	MoveL [[143.345,1275.593,0.000],[0.00000002,0.00000004,1.00000000,-0.00000004],[0,-1,0,0],rdkExtax], rdkSpeed, rdkZone, rdkTool, \WObj:=rdkWObj;
	MoveL [[133.284,1275.429,0.000],[0.00000002,0.00000004,1.00000000,-0.00000004],[0,-1,0,0],rdkExtax], rdkSpeed, rdkZone, rdkTool, \WObj:=rdkWObj;
	MoveL [[123.224,1275.245,0.000],[0.00000002,0.00000004,1.00000000,-0.00000004],[0,-1,0,0],rdkExtax], rdkSpeed, rdkZone, rdkTool, \WObj:=rdkWObj;
	MoveL [[113.164,1275.040,0.000],[0.00000002,0.00000004,1.00000000,-0.00000004],[0,-1,0,0],rdkExtax], rdkSpeed, rdkZone, rdkTool, \WObj:=rdkWObj;
	MoveL [[103.103,1274.816,0.000],[0.00000002,0.00000004,1.00000000,-0.00000004],[0,-1,0,0],rdkExtax], rdkSpeed, rdkZone, rdkTool, \WObj:=rdkWObj;
	MoveL [[93.043,1274.573,0.000],[0.00000002,0.00000004,1.00000000,-0.00000004],[0,-1,0,0],rdkExtax], rdkSpeed, rdkZone, rdkTool, \WObj:=rdkWObj;
	MoveL [[82.983,1274.311,0.000],[0.00000002,0.00000004,1.00000000,-0.00000004],[0,-1,0,0],rdkExtax], rdkSpeed, rdkZone, rdkTool, \WObj:=rdkWObj;
	MoveL [[72.922,1274.032,0.000],[0.00000002,0.00000004,1.00000000,-0.00000004],[0,-1,0,0],rdkExtax], rdkSpeed, rdkZone, rdkTool, \WObj:=rdkWObj;
	MoveL [[62.862,1273.736,0.000],[0.00000002,0.00000004,1.00000000,-0.00000004],[0,-1,0,0],rdkExtax], rdkSpeed, rdkZone, rdkTool, \WObj:=rdkWObj;
	MoveL [[52.801,1273.423,0.000],[0.00000002,0.00000004,1.00000000,-0.00000004],[0,-1,0,0],rdkExtax], rdkSpeed, rdkZone, rdkTool, \WObj:=rdkWObj;
	MoveL [[42.741,1273.094,0.000],[0.00000002,0.00000004,1.00000000,-0.00000004],[0,-1,0,0],rdkExtax], rdkSpeed, rdkZone, rdkTool, \WObj:=rdkWObj;
	MoveL [[32.680,1272.749,0.000],[0.00000002,0.00000004,1.00000000,-0.00000004],[0,-1,0,0],rdkExtax], rdkSpeed, rdkZone, rdkTool, \WObj:=rdkWObj;
	MoveL [[22.620,1272.390,0.000],[0.00000002,0.00000004,1.00000000,-0.00000004],[0,-1,0,0],rdkExtax], rdkSpeed, rdkZone, rdkTool, \WObj:=rdkWObj;
	MoveL [[16.560,1277.001,0.000],[0.00000002,0.00000004,1.00000000,-0.00000004],[0,-1,0,0],rdkExtax], rdkSpeed, rdkZone, rdkTool, \WObj:=rdkWObj;
	MoveL [[14.353,1286.214,0.000],[0.00000002,0.00000004,1.00000000,-0.00000004],[0,-1,0,0],rdkExtax], rdkSpeed, rdkZone, rdkTool, \WObj:=rdkWObj;
	MoveL [[12.501,1295.620,0.000],[0.00000002,0.00000004,1.00000000,-0.00000004],[0,-1,0,0],rdkExtax], rdkSpeed, rdkZone, rdkTool, \WObj:=rdkWObj;
	MoveL [[10.983,1305.202,0.000],[0.00000002,0.00000004,1.00000000,-0.00000004],[0,-1,0,0],rdkExtax], rdkSpeed, rdkZone, rdkTool, \WObj:=rdkWObj;
	MoveL [[9.778,1314.942,0.000],[0.00000002,0.00000004,1.00000000,-0.00000004],[0,-1,0,0],rdkExtax], rdkSpeed, rdkZone, rdkTool, \WObj:=rdkWObj;
	MoveL [[8.863,1324.822,0.000],[0.00000002,0.00000004,1.00000000,-0.00000004],[0,-1,0,0],rdkExtax], rdkSpeed, rdkZone, rdkTool, \WObj:=rdkWObj;
	MoveL [[8.219,1334.824,0.000],[0.00000002,0.00000004,1.00000000,-0.00000004],[0,-1,0,0],rdkExtax], rdkSpeed, rdkZone, rdkTool, \WObj:=rdkWObj;
	MoveL [[7.822,1344.931,0.000],[0.00000002,0.00000004,1.00000000,-0.00000004],[0,-1,0,0],rdkExtax], rdkSpeed, rdkZone, rdkTool, \WObj:=rdkWObj;
	MoveL [[7.652,1355.125,0.000],[0.00000002,0.00000004,1.00000000,-0.00000004],[0,-1,0,0],rdkExtax], rdkSpeed, rdkZone, rdkTool, \WObj:=rdkWObj;
	MoveL [[7.687,1365.387,0.000],[0.00000002,0.00000004,1.00000000,-0.00000004],[0,-1,0,0],rdkExtax], rdkSpeed, rdkZone, rdkTool, \WObj:=rdkWObj;
	MoveL [[7.907,1375.701,0.000],[0.00000002,0.00000004,1.00000000,-0.00000004],[0,-1,0,0],rdkExtax], rdkSpeed, rdkZone, rdkTool, \WObj:=rdkWObj;
	MoveL [[8.289,1386.047,0.000],[0.00000002,0.00000004,1.00000000,-0.00000004],[0,-1,0,0],rdkExtax], rdkSpeed, rdkZone, rdkTool, \WObj:=rdkWObj;
	MoveL [[8.812,1396.409,0.000],[0.00000002,0.00000004,1.00000000,-0.00000004],[0,-1,0,0],rdkExtax], rdkSpeed, rdkZone, rdkTool, \WObj:=rdkWObj;
	MoveL [[9.454,1406.769,0.000],[0.00000002,0.00000004,1.00000000,-0.00000004],[0,-1,0,0],rdkExtax], rdkSpeed, rdkZone, rdkTool, \WObj:=rdkWObj;
	MoveL [[10.195,1417.109,0.000],[0.00000002,0.00000004,1.00000000,-0.00000004],[0,-1,0,0],rdkExtax], rdkSpeed, rdkZone, rdkTool, \WObj:=rdkWObj;
	MoveL [[11.013,1427.410,0.000],[0.00000002,0.00000004,1.00000000,-0.00000004],[0,-1,0,0],rdkExtax], rdkSpeed, rdkZone, rdkTool, \WObj:=rdkWObj;
	MoveL [[11.886,1437.656,0.000],[0.00000002,0.00000004,1.00000000,-0.00000004],[0,-1,0,0],rdkExtax], rdkSpeed, rdkZone, rdkTool, \WObj:=rdkWObj;
	MoveL [[12.793,1447.828,0.000],[0.00000002,0.00000004,1.00000000,-0.00000004],[0,-1,0,0],rdkExtax], rdkSpeed, rdkZone, rdkTool, \WObj:=rdkWObj;
	MoveL [[13.713,1457.908,0.000],[0.00000002,0.00000004,1.00000000,-0.00000004],[0,-1,0,0],rdkExtax], rdkSpeed, rdkZone, rdkTool, \WObj:=rdkWObj;
	MoveL [[14.624,1467.879,0.000],[0.00000002,0.00000004,1.00000000,-0.00000004],[0,-1,0,0],rdkExtax], rdkSpeed, rdkZone, rdkTool, \WObj:=rdkWObj;
	MoveL [[15.505,1477.723,0.000],[0.00000002,0.00000004,1.00000000,-0.00000004],[0,-1,0,0],rdkExtax], rdkSpeed, rdkZone, rdkTool, \WObj:=rdkWObj;
	MoveL [[16.772,1487.917,0.000],[0.00000002,0.00000004,1.00000000,-0.00000004],[0,-1,0,0],rdkExtax], rdkSpeed, rdkZone, rdkTool, \WObj:=rdkWObj;
	MoveL [[18.876,1498.151,0.000],[0.00000002,0.00000004,1.00000000,-0.00000004],[0,-1,0,0],rdkExtax], rdkSpeed, rdkZone, rdkTool, \WObj:=rdkWObj;
	MoveL [[21.647,1508.050,0.000],[0.00000002,0.00000004,1.00000000,-0.00000004],[0,-1,0,0],rdkExtax], rdkSpeed, rdkZone, rdkTool, \WObj:=rdkWObj;
	MoveL [[25.057,1517.606,0.000],[0.00000002,0.00000004,1.00000000,-0.00000004],[0,-1,0,0],rdkExtax], rdkSpeed, rdkZone, rdkTool, \WObj:=rdkWObj;
	MoveL [[29.077,1526.811,0.000],[0.00000002,0.00000004,1.00000000,-0.00000004],[0,-1,0,0],rdkExtax], rdkSpeed, rdkZone, rdkTool, \WObj:=rdkWObj;
	MoveL [[33.677,1535.657,0.000],[0.00000002,0.00000004,1.00000000,-0.00000004],[0,-1,0,0],rdkExtax], rdkSpeed, rdkZone, rdkTool, \WObj:=rdkWObj;
	MoveL [[38.828,1544.135,0.000],[0.00000002,0.00000004,1.00000000,-0.00000004],[0,-1,0,0],rdkExtax], rdkSpeed, rdkZone, rdkTool, \WObj:=rdkWObj;
	MoveL [[44.502,1552.237,0.000],[0.00000002,0.00000004,1.00000000,-0.00000004],[0,-1,0,0],rdkExtax], rdkSpeed, rdkZone, rdkTool, \WObj:=rdkWObj;
	MoveL [[50.668,1559.956,0.000],[0.00000002,0.00000004,1.00000000,-0.00000004],[0,-1,0,0],rdkExtax], rdkSpeed, rdkZone, rdkTool, \WObj:=rdkWObj;
	MoveL [[57.299,1567.283,0.000],[0.00000002,0.00000004,1.00000000,-0.00000004],[0,-1,0,0],rdkExtax], rdkSpeed, rdkZone, rdkTool, \WObj:=rdkWObj;
	MoveL [[64.364,1574.209,0.000],[0.00000002,0.00000004,1.00000000,-0.00000004],[0,-1,0,0],rdkExtax], rdkSpeed, rdkZone, rdkTool, \WObj:=rdkWObj;
	MoveL [[71.835,1580.728,0.000],[0.00000002,0.00000004,1.00000000,-0.00000004],[0,-1,0,0],rdkExtax], rdkSpeed, rdkZone, rdkTool, \WObj:=rdkWObj;
	MoveL [[79.683,1586.830,0.000],[0.00000002,0.00000004,1.00000000,-0.00000004],[0,-1,0,0],rdkExtax], rdkSpeed, rdkZone, rdkTool, \WObj:=rdkWObj;
	MoveL [[87.878,1592.508,0.000],[0.00000002,0.00000004,1.00000000,-0.00000004],[0,-1,0,0],rdkExtax], rdkSpeed, rdkZone, rdkTool, \WObj:=rdkWObj;
	MoveL [[96.392,1597.753,0.000],[0.00000002,0.00000004,1.00000000,-0.00000004],[0,-1,0,0],rdkExtax], rdkSpeed, rdkZone, rdkTool, \WObj:=rdkWObj;
	MoveL [[105.194,1602.558,0.000],[0.00000002,0.00000004,1.00000000,-0.00000004],[0,-1,0,0],rdkExtax], rdkSpeed, rdkZone, rdkTool, \WObj:=rdkWObj;
	MoveL [[114.257,1606.914,0.000],[0.00000002,0.00000004,1.00000000,-0.00000004],[0,-1,0,0],rdkExtax], rdkSpeed, rdkZone, rdkTool, \WObj:=rdkWObj;
	MoveL [[123.551,1610.813,0.000],[0.00000002,0.00000004,1.00000000,-0.00000004],[0,-1,0,0],rdkExtax], rdkSpeed, rdkZone, rdkTool, \WObj:=rdkWObj;
	MoveL [[133.047,1614.246,0.000],[0.00000002,0.00000004,1.00000000,-0.00000004],[0,-1,0,0],rdkExtax], rdkSpeed, rdkZone, rdkTool, \WObj:=rdkWObj;
	MoveL [[142.716,1617.207,0.000],[0.00000002,0.00000004,1.00000000,-0.00000004],[0,-1,0,0],rdkExtax], rdkSpeed, rdkZone, rdkTool, \WObj:=rdkWObj;
	MoveL [[152.528,1619.686,0.000],[0.00000002,0.00000004,1.00000000,-0.00000004],[0,-1,0,0],rdkExtax], rdkSpeed, rdkZone, rdkTool, \WObj:=rdkWObj;
	MoveL [[162.454,1621.675,0.000],[0.00000002,0.00000004,1.00000000,-0.00000004],[0,-1,0,0],rdkExtax], rdkSpeed, rdkZone, rdkTool, \WObj:=rdkWObj;
	MoveL [[172.466,1623.167,0.000],[0.00000002,0.00000004,1.00000000,-0.00000004],[0,-1,0,0],rdkExtax], rdkSpeed, rdkZone, rdkTool, \WObj:=rdkWObj;
	MoveL [[182.535,1624.153,0.000],[0.00000002,0.00000004,1.00000000,-0.00000004],[0,-1,0,0],rdkExtax], rdkSpeed, rdkZone, rdkTool, \WObj:=rdkWObj;
	MoveL [[192.630,1624.625,0.000],[0.00000002,0.00000004,1.00000000,-0.00000004],[0,-1,0,0],rdkExtax], rdkSpeed, rdkZone, rdkTool, \WObj:=rdkWObj;
	MoveL [[191.948,1521.248,0.000],[0.00000002,0.00000004,1.00000000,-0.00000004],[0,-1,0,0],rdkExtax], rdkSpeed, rdkZone, rdkTool, \WObj:=rdkWObj;
	MoveL [[181.490,1520.957,0.000],[0.00000002,0.00000004,1.00000000,-0.00000004],[0,-1,0,0],rdkExtax], rdkSpeed, rdkZone, rdkTool, \WObj:=rdkWObj;
	MoveL [[171.373,1519.493,0.000],[0.00000002,0.00000004,1.00000000,-0.00000004],[0,-1,0,0],rdkExtax], rdkSpeed, rdkZone, rdkTool, \WObj:=rdkWObj;
	MoveL [[161.642,1516.933,0.000],[0.00000002,0.00000004,1.00000000,-0.00000004],[0,-1,0,0],rdkExtax], rdkSpeed, rdkZone, rdkTool, \WObj:=rdkWObj;
	MoveL [[152.344,1513.350,0.000],[0.00000002,0.00000004,1.00000000,-0.00000004],[0,-1,0,0],rdkExtax], rdkSpeed, rdkZone, rdkTool, \WObj:=rdkWObj;
	MoveL [[143.525,1508.821,0.000],[0.00000002,0.00000004,1.00000000,-0.00000004],[0,-1,0,0],rdkExtax], rdkSpeed, rdkZone, rdkTool, \WObj:=rdkWObj;
	MoveL [[135.231,1503.420,0.000],[0.00000002,0.00000004,1.00000000,-0.00000004],[0,-1,0,0],rdkExtax], rdkSpeed, rdkZone, rdkTool, \WObj:=rdkWObj;
	MoveL [[127.510,1497.222,0.000],[0.00000002,0.00000004,1.00000000,-0.00000004],[0,-1,0,0],rdkExtax], rdkSpeed, rdkZone, rdkTool, \WObj:=rdkWObj;
	MoveL [[120.406,1490.303,0.000],[0.00000002,0.00000004,1.00000000,-0.00000004],[0,-1,0,0],rdkExtax], rdkSpeed, rdkZone, rdkTool, \WObj:=rdkWObj;
	MoveL [[113.967,1482.738,0.000],[0.00000002,0.00000004,1.00000000,-0.00000004],[0,-1,0,0],rdkExtax], rdkSpeed, rdkZone, rdkTool, \WObj:=rdkWObj;
	MoveL [[108.239,1474.601,0.000],[0.00000002,0.00000004,1.00000000,-0.00000004],[0,-1,0,0],rdkExtax], rdkSpeed, rdkZone, rdkTool, \WObj:=rdkWObj;
	MoveL [[103.267,1465.968,0.000],[0.00000002,0.00000004,1.00000000,-0.00000004],[0,-1,0,0],rdkExtax], rdkSpeed, rdkZone, rdkTool, \WObj:=rdkWObj;
	MoveL [[99.099,1456.914,0.000],[0.00000002,0.00000004,1.00000000,-0.00000004],[0,-1,0,0],rdkExtax], rdkSpeed, rdkZone, rdkTool, \WObj:=rdkWObj;
	MoveL [[95.780,1447.514,0.000],[0.00000002,0.00000004,1.00000000,-0.00000004],[0,-1,0,0],rdkExtax], rdkSpeed, rdkZone, rdkTool, \WObj:=rdkWObj;
	MoveL [[93.357,1437.843,0.000],[0.00000002,0.00000004,1.00000000,-0.00000004],[0,-1,0,0],rdkExtax], rdkSpeed, rdkZone, rdkTool, \WObj:=rdkWObj;
	MoveL [[91.876,1427.977,0.000],[0.00000002,0.00000004,1.00000000,-0.00000004],[0,-1,0,0],rdkExtax], rdkSpeed, rdkZone, rdkTool, \WObj:=rdkWObj;
	MoveL [[91.384,1417.990,0.000],[0.00000002,0.00000004,1.00000000,-0.00000004],[0,-1,0,0],rdkExtax], rdkSpeed, rdkZone, rdkTool, \WObj:=rdkWObj;
	MoveL [[91.927,1407.958,0.000],[0.00000002,0.00000004,1.00000000,-0.00000004],[0,-1,0,0],rdkExtax], rdkSpeed, rdkZone, rdkTool, \WObj:=rdkWObj;
	MoveL [[93.550,1397.955,0.000],[0.00000002,0.00000004,1.00000000,-0.00000004],[0,-1,0,0],rdkExtax], rdkSpeed, rdkZone, rdkTool, \WObj:=rdkWObj;
	MoveL [[96.301,1388.057,0.000],[0.00000002,0.00000004,1.00000000,-0.00000004],[0,-1,0,0],rdkExtax], rdkSpeed, rdkZone, rdkTool, \WObj:=rdkWObj;
	MoveL [[101.782,1381.318,0.000],[0.00000002,0.00000004,1.00000000,-0.00000004],[0,-1,0,0],rdkExtax], rdkSpeed, rdkZone, rdkTool, \WObj:=rdkWObj;
	MoveL [[111.384,1381.237,0.000],[0.00000002,0.00000004,1.00000000,-0.00000004],[0,-1,0,0],rdkExtax], rdkSpeed, rdkZone, rdkTool, \WObj:=rdkWObj;
	MoveL [[121.241,1380.943,0.000],[0.00000002,0.00000004,1.00000000,-0.00000004],[0,-1,0,0],rdkExtax], rdkSpeed, rdkZone, rdkTool, \WObj:=rdkWObj;
	MoveL [[131.317,1380.480,0.000],[0.00000002,0.00000004,1.00000000,-0.00000004],[0,-1,0,0],rdkExtax], rdkSpeed, rdkZone, rdkTool, \WObj:=rdkWObj;
	MoveL [[141.577,1379.891,0.000],[0.00000002,0.00000004,1.00000000,-0.00000004],[0,-1,0,0],rdkExtax], rdkSpeed, rdkZone, rdkTool, \WObj:=rdkWObj;
	MoveL [[151.984,1379.219,0.000],[0.00000002,0.00000004,1.00000000,-0.00000004],[0,-1,0,0],rdkExtax], rdkSpeed, rdkZone, rdkTool, \WObj:=rdkWObj;
	MoveL [[162.504,1378.508,0.000],[0.00000002,0.00000004,1.00000000,-0.00000004],[0,-1,0,0],rdkExtax], rdkSpeed, rdkZone, rdkTool, \WObj:=rdkWObj;
	MoveL [[173.101,1377.802,0.000],[0.00000002,0.00000004,1.00000000,-0.00000004],[0,-1,0,0],rdkExtax], rdkSpeed, rdkZone, rdkTool, \WObj:=rdkWObj;
	MoveL [[183.740,1377.143,0.000],[0.00000002,0.00000004,1.00000000,-0.00000004],[0,-1,0,0],rdkExtax], rdkSpeed, rdkZone, rdkTool, \WObj:=rdkWObj;
	MoveL [[194.385,1376.575,0.000],[0.00000002,0.00000004,1.00000000,-0.00000004],[0,-1,0,0],rdkExtax], rdkSpeed, rdkZone, rdkTool, \WObj:=rdkWObj;
	MoveL [[205.000,1376.141,0.000],[0.00000002,0.00000004,1.00000000,-0.00000004],[0,-1,0,0],rdkExtax], rdkSpeed, rdkZone, rdkTool, \WObj:=rdkWObj;
	MoveL [[215.551,1375.885,0.000],[0.00000002,0.00000004,1.00000000,-0.00000004],[0,-1,0,0],rdkExtax], rdkSpeed, rdkZone, rdkTool, \WObj:=rdkWObj;
	MoveL [[226.001,1375.850,0.000],[0.00000002,0.00000004,1.00000000,-0.00000004],[0,-1,0,0],rdkExtax], rdkSpeed, rdkZone, rdkTool, \WObj:=rdkWObj;
	MoveL [[236.316,1376.080,0.000],[0.00000002,0.00000004,1.00000000,-0.00000004],[0,-1,0,0],rdkExtax], rdkSpeed, rdkZone, rdkTool, \WObj:=rdkWObj;
	MoveL [[246.459,1376.617,0.000],[0.00000002,0.00000004,1.00000000,-0.00000004],[0,-1,0,0],rdkExtax], rdkSpeed, rdkZone, rdkTool, \WObj:=rdkWObj;
	MoveL [[256.395,1377.506,0.000],[0.00000002,0.00000004,1.00000000,-0.00000004],[0,-1,0,0],rdkExtax], rdkSpeed, rdkZone, rdkTool, \WObj:=rdkWObj;
	MoveL [[266.090,1378.789,0.000],[0.00000002,0.00000004,1.00000000,-0.00000004],[0,-1,0,0],rdkExtax], rdkSpeed, rdkZone, rdkTool, \WObj:=rdkWObj;
	MoveL [[275.506,1380.510,0.000],[0.00000002,0.00000004,1.00000000,-0.00000004],[0,-1,0,0],rdkExtax], rdkSpeed, rdkZone, rdkTool, \WObj:=rdkWObj;
	MoveL [[284.610,1382.713,0.000],[0.00000002,0.00000004,1.00000000,-0.00000004],[0,-1,0,0],rdkExtax], rdkSpeed, rdkZone, rdkTool, \WObj:=rdkWObj;
	MoveL [[293.364,1385.440,0.000],[0.00000002,0.00000004,1.00000000,-0.00000004],[0,-1,0,0],rdkExtax], rdkSpeed, rdkZone, rdkTool, \WObj:=rdkWObj;
	MoveL [[301.735,1388.735,0.000],[0.00000002,0.00000004,1.00000000,-0.00000004],[0,-1,0,0],rdkExtax], rdkSpeed, rdkZone, rdkTool, \WObj:=rdkWObj;
	MoveL [[305.438,1397.949,0.000],[0.00000002,0.00000004,1.00000000,-0.00000004],[0,-1,0,0],rdkExtax], rdkSpeed, rdkZone, rdkTool, \WObj:=rdkWObj;
	MoveL [[307.003,1408.567,0.000],[0.00000002,0.00000004,1.00000000,-0.00000004],[0,-1,0,0],rdkExtax], rdkSpeed, rdkZone, rdkTool, \WObj:=rdkWObj;
	MoveL [[307.559,1419.010,0.000],[0.00000002,0.00000004,1.00000000,-0.00000004],[0,-1,0,0],rdkExtax], rdkSpeed, rdkZone, rdkTool, \WObj:=rdkWObj;
	MoveL [[307.145,1429.225,0.000],[0.00000002,0.00000004,1.00000000,-0.00000004],[0,-1,0,0],rdkExtax], rdkSpeed, rdkZone, rdkTool, \WObj:=rdkWObj;
	MoveL [[305.794,1439.164,0.000],[0.00000002,0.00000004,1.00000000,-0.00000004],[0,-1,0,0],rdkExtax], rdkSpeed, rdkZone, rdkTool, \WObj:=rdkWObj;
	MoveL [[303.543,1448.776,0.000],[0.00000002,0.00000004,1.00000000,-0.00000004],[0,-1,0,0],rdkExtax], rdkSpeed, rdkZone, rdkTool, \WObj:=rdkWObj;
	MoveL [[300.427,1458.011,0.000],[0.00000002,0.00000004,1.00000000,-0.00000004],[0,-1,0,0],rdkExtax], rdkSpeed, rdkZone, rdkTool, \WObj:=rdkWObj;
	MoveL [[296.482,1466.819,0.000],[0.00000002,0.00000004,1.00000000,-0.00000004],[0,-1,0,0],rdkExtax], rdkSpeed, rdkZone, rdkTool, \WObj:=rdkWObj;
	MoveL [[291.744,1475.149,0.000],[0.00000002,0.00000004,1.00000000,-0.00000004],[0,-1,0,0],rdkExtax], rdkSpeed, rdkZone, rdkTool, \WObj:=rdkWObj;
	MoveL [[286.249,1482.952,0.000],[0.00000002,0.00000004,1.00000000,-0.00000004],[0,-1,0,0],rdkExtax], rdkSpeed, rdkZone, rdkTool, \WObj:=rdkWObj;
	MoveL [[280.032,1490.176,0.000],[0.00000002,0.00000004,1.00000000,-0.00000004],[0,-1,0,0],rdkExtax], rdkSpeed, rdkZone, rdkTool, \WObj:=rdkWObj;
	MoveL [[273.129,1496.773,0.000],[0.00000002,0.00000004,1.00000000,-0.00000004],[0,-1,0,0],rdkExtax], rdkSpeed, rdkZone, rdkTool, \WObj:=rdkWObj;
	MoveL [[265.575,1502.691,0.000],[0.00000002,0.00000004,1.00000000,-0.00000004],[0,-1,0,0],rdkExtax], rdkSpeed, rdkZone, rdkTool, \WObj:=rdkWObj;
	MoveL [[257.407,1507.881,0.000],[0.00000002,0.00000004,1.00000000,-0.00000004],[0,-1,0,0],rdkExtax], rdkSpeed, rdkZone, rdkTool, \WObj:=rdkWObj;
	MoveL [[248.660,1512.292,0.000],[0.00000002,0.00000004,1.00000000,-0.00000004],[0,-1,0,0],rdkExtax], rdkSpeed, rdkZone, rdkTool, \WObj:=rdkWObj;
	MoveL [[239.369,1515.875,0.000],[0.00000002,0.00000004,1.00000000,-0.00000004],[0,-1,0,0],rdkExtax], rdkSpeed, rdkZone, rdkTool, \WObj:=rdkWObj;
	MoveL [[229.571,1518.578,0.000],[0.00000002,0.00000004,1.00000000,-0.00000004],[0,-1,0,0],rdkExtax], rdkSpeed, rdkZone, rdkTool, \WObj:=rdkWObj;
	MoveL [[219.301,1520.353,0.000],[0.00000002,0.00000004,1.00000000,-0.00000004],[0,-1,0,0],rdkExtax], rdkSpeed, rdkZone, rdkTool, \WObj:=rdkWObj;
	MoveL [[208.595,1521.148,0.000],[0.00000002,0.00000004,1.00000000,-0.00000004],[0,-1,0,0],rdkExtax], rdkSpeed, rdkZone, rdkTool, \WObj:=rdkWObj;
	MoveL [[197.489,1520.913,0.000],[0.00000002,0.00000004,1.00000000,-0.00000004],[0,-1,0,0],rdkExtax], rdkSpeed, rdkZone, rdkTool, \WObj:=rdkWObj;
	MoveL [[197.489,1520.913,100.000],[0.00000002,0.00000004,1.00000000,-0.00000004],[0,-1,0,0],rdkExtax], rdkSpeed, rdkZone, rdkTool, \WObj:=rdkWObj;
	MoveL [[374.392,2000.149,100.000],[0.00000002,0.00000004,1.00000000,-0.00000004],[0,-1,0,0],rdkExtax], rdkSpeed, rdkZone, rdkTool, \WObj:=rdkWObj;
	TPWrite "Drawing path3000";
	SetColorRGB(0.643,0.071,0.000);
	MoveL [[374.392,2000.149,0.000],[0.00000002,0.00000004,1.00000000,-0.00000004],[0,-1,0,0],rdkExtax], rdkSpeed, rdkZone, rdkTool, \WObj:=rdkWObj;
	MoveL [[380.983,1992.390,0.000],[0.00000002,0.00000004,1.00000000,-0.00000004],[0,-1,0,0],rdkExtax], rdkSpeed, rdkZone, rdkTool, \WObj:=rdkWObj;
	MoveL [[386.344,1984.065,0.000],[0.00000002,0.00000004,1.00000000,-0.00000004],[0,-1,0,0],rdkExtax], rdkSpeed, rdkZone, rdkTool, \WObj:=rdkWObj;
	MoveL [[390.508,1975.269,0.000],[0.00000002,0.00000004,1.00000000,-0.00000004],[0,-1,0,0],rdkExtax], rdkSpeed, rdkZone, rdkTool, \WObj:=rdkWObj;
	MoveL [[393.510,1966.101,0.000],[0.00000002,0.00000004,1.00000000,-0.00000004],[0,-1,0,0],rdkExtax], rdkSpeed, rdkZone, rdkTool, \WObj:=rdkWObj;
	MoveL [[395.384,1956.658,0.000],[0.00000002,0.00000004,1.00000000,-0.00000004],[0,-1,0,0],rdkExtax], rdkSpeed, rdkZone, rdkTool, \WObj:=rdkWObj;
	MoveL [[396.164,1947.037,0.000],[0.00000002,0.00000004,1.00000000,-0.00000004],[0,-1,0,0],rdkExtax], rdkSpeed, rdkZone, rdkTool, \WObj:=rdkWObj;
	MoveL [[395.885,1937.335,0.000],[0.00000002,0.00000004,1.00000000,-0.00000004],[0,-1,0,0],rdkExtax], rdkSpeed, rdkZone, rdkTool, \WObj:=rdkWObj;
	MoveL [[394.580,1927.650,0.000],[0.00000002,0.00000004,1.00000000,-0.00000004],[0,-1,0,0],rdkExtax], rdkSpeed, rdkZone, rdkTool, \WObj:=rdkWObj;
	MoveL [[392.283,1918.079,0.000],[0.00000002,0.00000004,1.00000000,-0.00000004],[0,-1,0,0],rdkExtax], rdkSpeed, rdkZone, rdkTool, \WObj:=rdkWObj;
	MoveL [[389.030,1908.719,0.000],[0.00000002,0.00000004,1.00000000,-0.00000004],[0,-1,0,0],rdkExtax], rdkSpeed, rdkZone, rdkTool, \WObj:=rdkWObj;
	MoveL [[384.853,1899.669,0.000],[0.00000002,0.00000004,1.00000000,-0.00000004],[0,-1,0,0],rdkExtax], rdkSpeed, rdkZone, rdkTool, \WObj:=rdkWObj;
	MoveL [[379.788,1891.024,0.000],[0.00000002,0.00000004,1.00000000,-0.00000004],[0,-1,0,0],rdkExtax], rdkSpeed, rdkZone, rdkTool, \WObj:=rdkWObj;
	MoveL [[373.868,1882.883,0.000],[0.00000002,0.00000004,1.00000000,-0.00000004],[0,-1,0,0],rdkExtax], rdkSpeed, rdkZone, rdkTool, \WObj:=rdkWObj;
	MoveL [[367.127,1875.342,0.000],[0.00000002,0.00000004,1.00000000,-0.00000004],[0,-1,0,0],rdkExtax], rdkSpeed, rdkZone, rdkTool, \WObj:=rdkWObj;
	MoveL [[359.601,1868.499,0.000],[0.00000002,0.00000004,1.00000000,-0.00000004],[0,-1,0,0],rdkExtax], rdkSpeed, rdkZone, rdkTool, \WObj:=rdkWObj;
	MoveL [[351.322,1862.452,0.000],[0.00000002,0.00000004,1.00000000,-0.00000004],[0,-1,0,0],rdkExtax], rdkSpeed, rdkZone, rdkTool, \WObj:=rdkWObj;
	MoveL [[342.325,1857.297,0.000],[0.00000002,0.00000004,1.00000000,-0.00000004],[0,-1,0,0],rdkExtax], rdkSpeed, rdkZone, rdkTool, \WObj:=rdkWObj;
	MoveL [[332.645,1853.133,0.000],[0.00000002,0.00000004,1.00000000,-0.00000004],[0,-1,0,0],rdkExtax], rdkSpeed, rdkZone, rdkTool, \WObj:=rdkWObj;
	MoveL [[322.314,1850.055,0.000],[0.00000002,0.00000004,1.00000000,-0.00000004],[0,-1,0,0],rdkExtax], rdkSpeed, rdkZone, rdkTool, \WObj:=rdkWObj;
	MoveL [[311.202,1847.909,0.000],[0.00000002,0.00000004,1.00000000,-0.00000004],[0,-1,0,0],rdkExtax], rdkSpeed, rdkZone, rdkTool, \WObj:=rdkWObj;
	MoveL [[299.905,1844.582,0.000],[0.00000002,0.00000004,1.00000000,-0.00000004],[0,-1,0,0],rdkExtax], rdkSpeed, rdkZone, rdkTool, \WObj:=rdkWObj;
	MoveL [[289.209,1839.822,0.000],[0.00000002,0.00000004,1.00000000,-0.00000004],[0,-1,0,0],rdkExtax], rdkSpeed, rdkZone, rdkTool, \WObj:=rdkWObj;
	MoveL [[279.340,1833.918,0.000],[0.00000002,0.00000004,1.00000000,-0.00000004],[0,-1,0,0],rdkExtax], rdkSpeed, rdkZone, rdkTool, \WObj:=rdkWObj;
	MoveL [[270.524,1827.156,0.000],[0.00000002,0.00000004,1.00000000,-0.00000004],[0,-1,0,0],rdkExtax], rdkSpeed, rdkZone, rdkTool, \WObj:=rdkWObj;
	MoveL [[262.987,1819.826,0.000],[0.00000002,0.00000004,1.00000000,-0.00000004],[0,-1,0,0],rdkExtax], rdkSpeed, rdkZone, rdkTool, \WObj:=rdkWObj;
	MoveL [[256.956,1812.214,0.000],[0.00000002,0.00000004,1.00000000,-0.00000004],[0,-1,0,0],rdkExtax], rdkSpeed, rdkZone, rdkTool, \WObj:=rdkWObj;
	MoveL [[252.657,1804.611,0.000],[0.00000002,0.00000004,1.00000000,-0.00000004],[0,-1,0,0],rdkExtax], rdkSpeed, rdkZone, rdkTool, \WObj:=rdkWObj;
	MoveL [[250.316,1797.302,0.000],[0.00000002,0.00000004,1.00000000,-0.00000004],[0,-1,0,0],rdkExtax], rdkSpeed, rdkZone, rdkTool, \WObj:=rdkWObj;
	MoveL [[250.159,1790.578,0.000],[0.00000002,0.00000004,1.00000000,-0.00000004],[0,-1,0,0],rdkExtax], rdkSpeed, rdkZone, rdkTool, \WObj:=rdkWObj;
	MoveL [[252.412,1784.725,0.000],[0.00000002,0.00000004,1.00000000,-0.00000004],[0,-1,0,0],rdkExtax], rdkSpeed, rdkZone, rdkTool, \WObj:=rdkWObj;
	MoveL [[257.302,1780.031,0.000],[0.00000002,0.00000004,1.00000000,-0.00000004],[0,-1,0,0],rdkExtax], rdkSpeed, rdkZone, rdkTool, \WObj:=rdkWObj;
	MoveL [[265.055,1776.786,0.000],[0.00000002,0.00000004,1.00000000,-0.00000004],[0,-1,0,0],rdkExtax], rdkSpeed, rdkZone, rdkTool, \WObj:=rdkWObj;
	MoveL [[275.896,1775.276,0.000],[0.00000002,0.00000004,1.00000000,-0.00000004],[0,-1,0,0],rdkExtax], rdkSpeed, rdkZone, rdkTool, \WObj:=rdkWObj;
	MoveL [[290.052,1775.790,0.000],[0.00000002,0.00000004,1.00000000,-0.00000004],[0,-1,0,0],rdkExtax], rdkSpeed, rdkZone, rdkTool, \WObj:=rdkWObj;
	MoveL [[303.834,1777.432,0.000],[0.00000002,0.00000004,1.00000000,-0.00000004],[0,-1,0,0],rdkExtax], rdkSpeed, rdkZone, rdkTool, \WObj:=rdkWObj;
	MoveL [[314.296,1778.411,0.000],[0.00000002,0.00000004,1.00000000,-0.00000004],[0,-1,0,0],rdkExtax], rdkSpeed, rdkZone, rdkTool, \WObj:=rdkWObj;
	MoveL [[325.048,1779.340,0.000],[0.00000002,0.00000004,1.00000000,-0.00000004],[0,-1,0,0],rdkExtax], rdkSpeed, rdkZone, rdkTool, \WObj:=rdkWObj;
	MoveL [[335.852,1780.022,0.000],[0.00000002,0.00000004,1.00000000,-0.00000004],[0,-1,0,0],rdkExtax], rdkSpeed, rdkZone, rdkTool, \WObj:=rdkWObj;
	MoveL [[346.467,1780.260,0.000],[0.00000002,0.00000004,1.00000000,-0.00000004],[0,-1,0,0],rdkExtax], rdkSpeed, rdkZone, rdkTool, \WObj:=rdkWObj;
	MoveL [[356.655,1779.857,0.000],[0.00000002,0.00000004,1.00000000,-0.00000004],[0,-1,0,0],rdkExtax], rdkSpeed, rdkZone, rdkTool, \WObj:=rdkWObj;
	MoveL [[366.177,1778.616,0.000],[0.00000002,0.00000004,1.00000000,-0.00000004],[0,-1,0,0],rdkExtax], rdkSpeed, rdkZone, rdkTool, \WObj:=rdkWObj;
	MoveL [[374.793,1776.339,0.000],[0.00000002,0.00000004,1.00000000,-0.00000004],[0,-1,0,0],rdkExtax], rdkSpeed, rdkZone, rdkTool, \WObj:=rdkWObj;
	MoveL [[382.264,1772.830,0.000],[0.00000002,0.00000004,1.00000000,-0.00000004],[0,-1,0,0],rdkExtax], rdkSpeed, rdkZone, rdkTool, \WObj:=rdkWObj;
	MoveL [[388.351,1767.892,0.000],[0.00000002,0.00000004,1.00000000,-0.00000004],[0,-1,0,0],rdkExtax], rdkSpeed, rdkZone, rdkTool, \WObj:=rdkWObj;
	MoveL [[392.816,1761.327,0.000],[0.00000002,0.00000004,1.00000000,-0.00000004],[0,-1,0,0],rdkExtax], rdkSpeed, rdkZone, rdkTool, \WObj:=rdkWObj;
	MoveL [[395.418,1752.940,0.000],[0.00000002,0.00000004,1.00000000,-0.00000004],[0,-1,0,0],rdkExtax], rdkSpeed, rdkZone, rdkTool, \WObj:=rdkWObj;
	MoveL [[395.918,1742.532,0.000],[0.00000002,0.00000004,1.00000000,-0.00000004],[0,-1,0,0],rdkExtax], rdkSpeed, rdkZone, rdkTool, \WObj:=rdkWObj;
	MoveL [[394.078,1729.906,0.000],[0.00000002,0.00000004,1.00000000,-0.00000004],[0,-1,0,0],rdkExtax], rdkSpeed, rdkZone, rdkTool, \WObj:=rdkWObj;
	MoveL [[392.731,1715.600,0.000],[0.00000002,0.00000004,1.00000000,-0.00000004],[0,-1,0,0],rdkExtax], rdkSpeed, rdkZone, rdkTool, \WObj:=rdkWObj;
	MoveL [[393.844,1703.189,0.000],[0.00000002,0.00000004,1.00000000,-0.00000004],[0,-1,0,0],rdkExtax], rdkSpeed, rdkZone, rdkTool, \WObj:=rdkWObj;
	MoveL [[393.047,1692.845,0.000],[0.00000002,0.00000004,1.00000000,-0.00000004],[0,-1,0,0],rdkExtax], rdkSpeed, rdkZone, rdkTool, \WObj:=rdkWObj;
	MoveL [[390.495,1684.403,0.000],[0.00000002,0.00000004,1.00000000,-0.00000004],[0,-1,0,0],rdkExtax], rdkSpeed, rdkZone, rdkTool, \WObj:=rdkWObj;
	MoveL [[386.347,1677.698,0.000],[0.00000002,0.00000004,1.00000000,-0.00000004],[0,-1,0,0],rdkExtax], rdkSpeed, rdkZone, rdkTool, \WObj:=rdkWObj;
	MoveL [[380.758,1672.565,0.000],[0.00000002,0.00000004,1.00000000,-0.00000004],[0,-1,0,0],rdkExtax], rdkSpeed, rdkZone, rdkTool, \WObj:=rdkWObj;
	MoveL [[373.886,1668.838,0.000],[0.00000002,0.00000004,1.00000000,-0.00000004],[0,-1,0,0],rdkExtax], rdkSpeed, rdkZone, rdkTool, \WObj:=rdkWObj;
	MoveL [[365.887,1666.354,0.000],[0.00000002,0.00000004,1.00000000,-0.00000004],[0,-1,0,0],rdkExtax], rdkSpeed, rdkZone, rdkTool, \WObj:=rdkWObj;
	MoveL [[356.917,1664.946,0.000],[0.00000002,0.00000004,1.00000000,-0.00000004],[0,-1,0,0],rdkExtax], rdkSpeed, rdkZone, rdkTool, \WObj:=rdkWObj;
	MoveL [[347.135,1664.451,0.000],[0.00000002,0.00000004,1.00000000,-0.00000004],[0,-1,0,0],rdkExtax], rdkSpeed, rdkZone, rdkTool, \WObj:=rdkWObj;
	MoveL [[336.696,1664.702,0.000],[0.00000002,0.00000004,1.00000000,-0.00000004],[0,-1,0,0],rdkExtax], rdkSpeed, rdkZone, rdkTool, \WObj:=rdkWObj;
	MoveL [[325.758,1665.535,0.000],[0.00000002,0.00000004,1.00000000,-0.00000004],[0,-1,0,0],rdkExtax], rdkSpeed, rdkZone, rdkTool, \WObj:=rdkWObj;
	MoveL [[314.476,1666.785,0.000],[0.00000002,0.00000004,1.00000000,-0.00000004],[0,-1,0,0],rdkExtax], rdkSpeed, rdkZone, rdkTool, \WObj:=rdkWObj;
	MoveL [[303.008,1668.286,0.000],[0.00000002,0.00000004,1.00000000,-0.00000004],[0,-1,0,0],rdkExtax], rdkSpeed, rdkZone, rdkTool, \WObj:=rdkWObj;
	MoveL [[291.511,1669.874,0.000],[0.00000002,0.00000004,1.00000000,-0.00000004],[0,-1,0,0],rdkExtax], rdkSpeed, rdkZone, rdkTool, \WObj:=rdkWObj;
	MoveL [[280.141,1671.384,0.000],[0.00000002,0.00000004,1.00000000,-0.00000004],[0,-1,0,0],rdkExtax], rdkSpeed, rdkZone, rdkTool, \WObj:=rdkWObj;
	MoveL [[269.055,1672.650,0.000],[0.00000002,0.00000004,1.00000000,-0.00000004],[0,-1,0,0],rdkExtax], rdkSpeed, rdkZone, rdkTool, \WObj:=rdkWObj;
	MoveL [[258.410,1673.508,0.000],[0.00000002,0.00000004,1.00000000,-0.00000004],[0,-1,0,0],rdkExtax], rdkSpeed, rdkZone, rdkTool, \WObj:=rdkWObj;
	MoveL [[248.363,1673.792,0.000],[0.00000002,0.00000004,1.00000000,-0.00000004],[0,-1,0,0],rdkExtax], rdkSpeed, rdkZone, rdkTool, \WObj:=rdkWObj;
	MoveL [[239.070,1673.338,0.000],[0.00000002,0.00000004,1.00000000,-0.00000004],[0,-1,0,0],rdkExtax], rdkSpeed, rdkZone, rdkTool, \WObj:=rdkWObj;
	MoveL [[230.688,1671.981,0.000],[0.00000002,0.00000004,1.00000000,-0.00000004],[0,-1,0,0],rdkExtax], rdkSpeed, rdkZone, rdkTool, \WObj:=rdkWObj;
	MoveL [[220.678,1672.266,0.000],[0.00000002,0.00000004,1.00000000,-0.00000004],[0,-1,0,0],rdkExtax], rdkSpeed, rdkZone, rdkTool, \WObj:=rdkWObj;
	MoveL [[210.627,1672.439,0.000],[0.00000002,0.00000004,1.00000000,-0.00000004],[0,-1,0,0],rdkExtax], rdkSpeed, rdkZone, rdkTool, \WObj:=rdkWObj;
	MoveL [[200.572,1672.480,0.000],[0.00000002,0.00000004,1.00000000,-0.00000004],[0,-1,0,0],rdkExtax], rdkSpeed, rdkZone, rdkTool, \WObj:=rdkWObj;
	MoveL [[190.513,1672.402,0.000],[0.00000002,0.00000004,1.00000000,-0.00000004],[0,-1,0,0],rdkExtax], rdkSpeed, rdkZone, rdkTool, \WObj:=rdkWObj;
	MoveL [[180.452,1672.223,0.000],[0.00000002,0.00000004,1.00000000,-0.00000004],[0,-1,0,0],rdkExtax], rdkSpeed, rdkZone, rdkTool, \WObj:=rdkWObj;
	MoveL [[170.388,1671.956,0.000],[0.00000002,0.00000004,1.00000000,-0.00000004],[0,-1,0,0],rdkExtax], rdkSpeed, rdkZone, rdkTool, \WObj:=rdkWObj;
	MoveL [[160.323,1671.617,0.000],[0.00000002,0.00000004,1.00000000,-0.00000004],[0,-1,0,0],rdkExtax], rdkSpeed, rdkZone, rdkTool, \WObj:=rdkWObj;
	MoveL [[150.258,1671.223,0.000],[0.00000002,0.00000004,1.00000000,-0.00000004],[0,-1,0,0],rdkExtax], rdkSpeed, rdkZone, rdkTool, \WObj:=rdkWObj;
	MoveL [[140.193,1670.787,0.000],[0.00000002,0.00000004,1.00000000,-0.00000004],[0,-1,0,0],rdkExtax], rdkSpeed, rdkZone, rdkTool, \WObj:=rdkWObj;
	MoveL [[130.128,1670.327,0.000],[0.00000002,0.00000004,1.00000000,-0.00000004],[0,-1,0,0],rdkExtax], rdkSpeed, rdkZone, rdkTool, \WObj:=rdkWObj;
	MoveL [[120.066,1669.856,0.000],[0.00000002,0.00000004,1.00000000,-0.00000004],[0,-1,0,0],rdkExtax], rdkSpeed, rdkZone, rdkTool, \WObj:=rdkWObj;
	MoveL [[110.006,1669.390,0.000],[0.00000002,0.00000004,1.00000000,-0.00000004],[0,-1,0,0],rdkExtax], rdkSpeed, rdkZone, rdkTool, \WObj:=rdkWObj;
	MoveL [[99.949,1668.946,0.000],[0.00000002,0.00000004,1.00000000,-0.00000004],[0,-1,0,0],rdkExtax], rdkSpeed, rdkZone, rdkTool, \WObj:=rdkWObj;
	MoveL [[89.897,1668.537,0.000],[0.00000002,0.00000004,1.00000000,-0.00000004],[0,-1,0,0],rdkExtax], rdkSpeed, rdkZone, rdkTool, \WObj:=rdkWObj;
	MoveL [[79.849,1668.180,0.000],[0.00000002,0.00000004,1.00000000,-0.00000004],[0,-1,0,0],rdkExtax], rdkSpeed, rdkZone, rdkTool, \WObj:=rdkWObj;
	MoveL [[69.808,1667.890,0.000],[0.00000002,0.00000004,1.00000000,-0.00000004],[0,-1,0,0],rdkExtax], rdkSpeed, rdkZone, rdkTool, \WObj:=rdkWObj;
	MoveL [[59.772,1667.683,0.000],[0.00000002,0.00000004,1.00000000,-0.00000004],[0,-1,0,0],rdkExtax], rdkSpeed, rdkZone, rdkTool, \WObj:=rdkWObj;
	MoveL [[49.744,1667.573,0.000],[0.00000002,0.00000004,1.00000000,-0.00000004],[0,-1,0,0],rdkExtax], rdkSpeed, rdkZone, rdkTool, \WObj:=rdkWObj;
	MoveL [[39.724,1667.576,0.000],[0.00000002,0.00000004,1.00000000,-0.00000004],[0,-1,0,0],rdkExtax], rdkSpeed, rdkZone, rdkTool, \WObj:=rdkWObj;
	MoveL [[29.712,1667.708,0.000],[0.00000002,0.00000004,1.00000000,-0.00000004],[0,-1,0,0],rdkExtax], rdkSpeed, rdkZone, rdkTool, \WObj:=rdkWObj;
	MoveL [[19.710,1667.983,0.000],[0.00000002,0.00000004,1.00000000,-0.00000004],[0,-1,0,0],rdkExtax], rdkSpeed, rdkZone, rdkTool, \WObj:=rdkWObj;
	MoveL [[11.076,1669.486,0.000],[0.00000002,0.00000004,1.00000000,-0.00000004],[0,-1,0,0],rdkExtax], rdkSpeed, rdkZone, rdkTool, \WObj:=rdkWObj;
	MoveL [[11.476,1679.058,0.000],[0.00000002,0.00000004,1.00000000,-0.00000004],[0,-1,0,0],rdkExtax], rdkSpeed, rdkZone, rdkTool, \WObj:=rdkWObj;
	MoveL [[11.234,1689.394,0.000],[0.00000002,0.00000004,1.00000000,-0.00000004],[0,-1,0,0],rdkExtax], rdkSpeed, rdkZone, rdkTool, \WObj:=rdkWObj;
	MoveL [[10.581,1700.248,0.000],[0.00000002,0.00000004,1.00000000,-0.00000004],[0,-1,0,0],rdkExtax], rdkSpeed, rdkZone, rdkTool, \WObj:=rdkWObj;
	MoveL [[9.744,1711.372,0.000],[0.00000002,0.00000004,1.00000000,-0.00000004],[0,-1,0,0],rdkExtax], rdkSpeed, rdkZone, rdkTool, \WObj:=rdkWObj;
	MoveL [[8.953,1722.520,0.000],[0.00000002,0.00000004,1.00000000,-0.00000004],[0,-1,0,0],rdkExtax], rdkSpeed, rdkZone, rdkTool, \WObj:=rdkWObj;
	MoveL [[8.437,1733.445,0.000],[0.00000002,0.00000004,1.00000000,-0.00000004],[0,-1,0,0],rdkExtax], rdkSpeed, rdkZone, rdkTool, \WObj:=rdkWObj;
	MoveL [[8.424,1743.901,0.000],[0.00000002,0.00000004,1.00000000,-0.00000004],[0,-1,0,0],rdkExtax], rdkSpeed, rdkZone, rdkTool, \WObj:=rdkWObj;
	MoveL [[9.145,1753.640,0.000],[0.00000002,0.00000004,1.00000000,-0.00000004],[0,-1,0,0],rdkExtax], rdkSpeed, rdkZone, rdkTool, \WObj:=rdkWObj;
	MoveL [[10.827,1762.417,0.000],[0.00000002,0.00000004,1.00000000,-0.00000004],[0,-1,0,0],rdkExtax], rdkSpeed, rdkZone, rdkTool, \WObj:=rdkWObj;
	MoveL [[13.700,1769.983,0.000],[0.00000002,0.00000004,1.00000000,-0.00000004],[0,-1,0,0],rdkExtax], rdkSpeed, rdkZone, rdkTool, \WObj:=rdkWObj;
	MoveL [[17.992,1776.092,0.000],[0.00000002,0.00000004,1.00000000,-0.00000004],[0,-1,0,0],rdkExtax], rdkSpeed, rdkZone, rdkTool, \WObj:=rdkWObj;
	MoveL [[23.934,1780.498,0.000],[0.00000002,0.00000004,1.00000000,-0.00000004],[0,-1,0,0],rdkExtax], rdkSpeed, rdkZone, rdkTool, \WObj:=rdkWObj;
	MoveL [[31.753,1782.954,0.000],[0.00000002,0.00000004,1.00000000,-0.00000004],[0,-1,0,0],rdkExtax], rdkSpeed, rdkZone, rdkTool, \WObj:=rdkWObj;
	MoveL [[41.679,1783.213,0.000],[0.00000002,0.00000004,1.00000000,-0.00000004],[0,-1,0,0],rdkExtax], rdkSpeed, rdkZone, rdkTool, \WObj:=rdkWObj;
	MoveL [[53.941,1781.028,0.000],[0.00000002,0.00000004,1.00000000,-0.00000004],[0,-1,0,0],rdkExtax], rdkSpeed, rdkZone, rdkTool, \WObj:=rdkWObj;
	MoveL [[67.287,1777.073,0.000],[0.00000002,0.00000004,1.00000000,-0.00000004],[0,-1,0,0],rdkExtax], rdkSpeed, rdkZone, rdkTool, \WObj:=rdkWObj;
	MoveL [[77.310,1775.346,0.000],[0.00000002,0.00000004,1.00000000,-0.00000004],[0,-1,0,0],rdkExtax], rdkSpeed, rdkZone, rdkTool, \WObj:=rdkWObj;
	MoveL [[87.999,1774.101,0.000],[0.00000002,0.00000004,1.00000000,-0.00000004],[0,-1,0,0],rdkExtax], rdkSpeed, rdkZone, rdkTool, \WObj:=rdkWObj;
	MoveL [[99.025,1773.424,0.000],[0.00000002,0.00000004,1.00000000,-0.00000004],[0,-1,0,0],rdkExtax], rdkSpeed, rdkZone, rdkTool, \WObj:=rdkWObj;
	MoveL [[110.061,1773.401,0.000],[0.00000002,0.00000004,1.00000000,-0.00000004],[0,-1,0,0],rdkExtax], rdkSpeed, rdkZone, rdkTool, \WObj:=rdkWObj;
	MoveL [[120.779,1774.121,0.000],[0.00000002,0.00000004,1.00000000,-0.00000004],[0,-1,0,0],rdkExtax], rdkSpeed, rdkZone, rdkTool, \WObj:=rdkWObj;
	MoveL [[130.849,1775.668,0.000],[0.00000002,0.00000004,1.00000000,-0.00000004],[0,-1,0,0],rdkExtax], rdkSpeed, rdkZone, rdkTool, \WObj:=rdkWObj;
	MoveL [[139.945,1778.131,0.000],[0.00000002,0.00000004,1.00000000,-0.00000004],[0,-1,0,0],rdkExtax], rdkSpeed, rdkZone, rdkTool, \WObj:=rdkWObj;
	MoveL [[147.737,1781.595,0.000],[0.00000002,0.00000004,1.00000000,-0.00000004],[0,-1,0,0],rdkExtax], rdkSpeed, rdkZone, rdkTool, \WObj:=rdkWObj;
	MoveL [[153.898,1786.148,0.000],[0.00000002,0.00000004,1.00000000,-0.00000004],[0,-1,0,0],rdkExtax], rdkSpeed, rdkZone, rdkTool, \WObj:=rdkWObj;
	MoveL [[158.099,1791.876,0.000],[0.00000002,0.00000004,1.00000000,-0.00000004],[0,-1,0,0],rdkExtax], rdkSpeed, rdkZone, rdkTool, \WObj:=rdkWObj;
	MoveL [[160.012,1798.866,0.000],[0.00000002,0.00000004,1.00000000,-0.00000004],[0,-1,0,0],rdkExtax], rdkSpeed, rdkZone, rdkTool, \WObj:=rdkWObj;
	MoveL [[159.309,1807.205,0.000],[0.00000002,0.00000004,1.00000000,-0.00000004],[0,-1,0,0],rdkExtax], rdkSpeed, rdkZone, rdkTool, \WObj:=rdkWObj;
	MoveL [[155.661,1816.979,0.000],[0.00000002,0.00000004,1.00000000,-0.00000004],[0,-1,0,0],rdkExtax], rdkSpeed, rdkZone, rdkTool, \WObj:=rdkWObj;
	MoveL [[148.741,1828.275,0.000],[0.00000002,0.00000004,1.00000000,-0.00000004],[0,-1,0,0],rdkExtax], rdkSpeed, rdkZone, rdkTool, \WObj:=rdkWObj;
	MoveL [[139.475,1839.503,0.000],[0.00000002,0.00000004,1.00000000,-0.00000004],[0,-1,0,0],rdkExtax], rdkSpeed, rdkZone, rdkTool, \WObj:=rdkWObj;
	MoveL [[132.032,1845.628,0.000],[0.00000002,0.00000004,1.00000000,-0.00000004],[0,-1,0,0],rdkExtax], rdkSpeed, rdkZone, rdkTool, \WObj:=rdkWObj;
	MoveL [[123.710,1850.978,0.000],[0.00000002,0.00000004,1.00000000,-0.00000004],[0,-1,0,0],rdkExtax], rdkSpeed, rdkZone, rdkTool, \WObj:=rdkWObj;
	MoveL [[114.674,1855.681,0.000],[0.00000002,0.00000004,1.00000000,-0.00000004],[0,-1,0,0],rdkExtax], rdkSpeed, rdkZone, rdkTool, \WObj:=rdkWObj;
	MoveL [[105.091,1859.864,0.000],[0.00000002,0.00000004,1.00000000,-0.00000004],[0,-1,0,0],rdkExtax], rdkSpeed, rdkZone, rdkTool, \WObj:=rdkWObj;
	MoveL [[95.124,1863.656,0.000],[0.00000002,0.00000004,1.00000000,-0.00000004],[0,-1,0,0],rdkExtax], rdkSpeed, rdkZone, rdkTool, \WObj:=rdkWObj;
	MoveL [[84.941,1867.185,0.000],[0.00000002,0.00000004,1.00000000,-0.00000004],[0,-1,0,0],rdkExtax], rdkSpeed, rdkZone, rdkTool, \WObj:=rdkWObj;
	MoveL [[74.706,1870.579,0.000],[0.00000002,0.00000004,1.00000000,-0.00000004],[0,-1,0,0],rdkExtax], rdkSpeed, rdkZone, rdkTool, \WObj:=rdkWObj;
	MoveL [[64.585,1873.965,0.000],[0.00000002,0.00000004,1.00000000,-0.00000004],[0,-1,0,0],rdkExtax], rdkSpeed, rdkZone, rdkTool, \WObj:=rdkWObj;
	MoveL [[54.744,1877.473,0.000],[0.00000002,0.00000004,1.00000000,-0.00000004],[0,-1,0,0],rdkExtax], rdkSpeed, rdkZone, rdkTool, \WObj:=rdkWObj;
	MoveL [[45.348,1881.228,0.000],[0.00000002,0.00000004,1.00000000,-0.00000004],[0,-1,0,0],rdkExtax], rdkSpeed, rdkZone, rdkTool, \WObj:=rdkWObj;
	MoveL [[36.562,1885.361,0.000],[0.00000002,0.00000004,1.00000000,-0.00000004],[0,-1,0,0],rdkExtax], rdkSpeed, rdkZone, rdkTool, \WObj:=rdkWObj;
	MoveL [[28.552,1889.999,0.000],[0.00000002,0.00000004,1.00000000,-0.00000004],[0,-1,0,0],rdkExtax], rdkSpeed, rdkZone, rdkTool, \WObj:=rdkWObj;
	MoveL [[21.484,1895.269,0.000],[0.00000002,0.00000004,1.00000000,-0.00000004],[0,-1,0,0],rdkExtax], rdkSpeed, rdkZone, rdkTool, \WObj:=rdkWObj;
	MoveL [[15.523,1901.300,0.000],[0.00000002,0.00000004,1.00000000,-0.00000004],[0,-1,0,0],rdkExtax], rdkSpeed, rdkZone, rdkTool, \WObj:=rdkWObj;
	MoveL [[10.835,1908.220,0.000],[0.00000002,0.00000004,1.00000000,-0.00000004],[0,-1,0,0],rdkExtax], rdkSpeed, rdkZone, rdkTool, \WObj:=rdkWObj;
	MoveL [[7.585,1916.156,0.000],[0.00000002,0.00000004,1.00000000,-0.00000004],[0,-1,0,0],rdkExtax], rdkSpeed, rdkZone, rdkTool, \WObj:=rdkWObj;
	MoveL [[5.939,1925.237,0.000],[0.00000002,0.00000004,1.00000000,-0.00000004],[0,-1,0,0],rdkExtax], rdkSpeed, rdkZone, rdkTool, \WObj:=rdkWObj;
	MoveL [[6.062,1935.591,0.000],[0.00000002,0.00000004,1.00000000,-0.00000004],[0,-1,0,0],rdkExtax], rdkSpeed, rdkZone, rdkTool, \WObj:=rdkWObj;
	MoveL [[8.119,1947.346,0.000],[0.00000002,0.00000004,1.00000000,-0.00000004],[0,-1,0,0],rdkExtax], rdkSpeed, rdkZone, rdkTool, \WObj:=rdkWObj;
	MoveL [[10.508,1960.470,0.000],[0.00000002,0.00000004,1.00000000,-0.00000004],[0,-1,0,0],rdkExtax], rdkSpeed, rdkZone, rdkTool, \WObj:=rdkWObj;
	MoveL [[10.150,1971.989,0.000],[0.00000002,0.00000004,1.00000000,-0.00000004],[0,-1,0,0],rdkExtax], rdkSpeed, rdkZone, rdkTool, \WObj:=rdkWObj;
	MoveL [[11.834,1980.898,0.000],[0.00000002,0.00000004,1.00000000,-0.00000004],[0,-1,0,0],rdkExtax], rdkSpeed, rdkZone, rdkTool, \WObj:=rdkWObj;
	MoveL [[15.364,1987.411,0.000],[0.00000002,0.00000004,1.00000000,-0.00000004],[0,-1,0,0],rdkExtax], rdkSpeed, rdkZone, rdkTool, \WObj:=rdkWObj;
	MoveL [[20.540,1991.739,0.000],[0.00000002,0.00000004,1.00000000,-0.00000004],[0,-1,0,0],rdkExtax], rdkSpeed, rdkZone, rdkTool, \WObj:=rdkWObj;
	MoveL [[27.164,1994.095,0.000],[0.00000002,0.00000004,1.00000000,-0.00000004],[0,-1,0,0],rdkExtax], rdkSpeed, rdkZone, rdkTool, \WObj:=rdkWObj;
	MoveL [[35.038,1994.692,0.000],[0.00000002,0.00000004,1.00000000,-0.00000004],[0,-1,0,0],rdkExtax], rdkSpeed, rdkZone, rdkTool, \WObj:=rdkWObj;
	MoveL [[43.961,1993.742,0.000],[0.00000002,0.00000004,1.00000000,-0.00000004],[0,-1,0,0],rdkExtax], rdkSpeed, rdkZone, rdkTool, \WObj:=rdkWObj;
	MoveL [[53.737,1991.458,0.000],[0.00000002,0.00000004,1.00000000,-0.00000004],[0,-1,0,0],rdkExtax], rdkSpeed, rdkZone, rdkTool, \WObj:=rdkWObj;
	MoveL [[64.167,1988.053,0.000],[0.00000002,0.00000004,1.00000000,-0.00000004],[0,-1,0,0],rdkExtax], rdkSpeed, rdkZone, rdkTool, \WObj:=rdkWObj;
	MoveL [[75.051,1983.738,0.000],[0.00000002,0.00000004,1.00000000,-0.00000004],[0,-1,0,0],rdkExtax], rdkSpeed, rdkZone, rdkTool, \WObj:=rdkWObj;
	MoveL [[86.191,1978.728,0.000],[0.00000002,0.00000004,1.00000000,-0.00000004],[0,-1,0,0],rdkExtax], rdkSpeed, rdkZone, rdkTool, \WObj:=rdkWObj;
	MoveL [[97.388,1973.233,0.000],[0.00000002,0.00000004,1.00000000,-0.00000004],[0,-1,0,0],rdkExtax], rdkSpeed, rdkZone, rdkTool, \WObj:=rdkWObj;
	MoveL [[108.445,1967.467,0.000],[0.00000002,0.00000004,1.00000000,-0.00000004],[0,-1,0,0],rdkExtax], rdkSpeed, rdkZone, rdkTool, \WObj:=rdkWObj;
	MoveL [[119.162,1961.643,0.000],[0.00000002,0.00000004,1.00000000,-0.00000004],[0,-1,0,0],rdkExtax], rdkSpeed, rdkZone, rdkTool, \WObj:=rdkWObj;
	MoveL [[129.340,1955.972,0.000],[0.00000002,0.00000004,1.00000000,-0.00000004],[0,-1,0,0],rdkExtax], rdkSpeed, rdkZone, rdkTool, \WObj:=rdkWObj;
	MoveL [[138.782,1950.668,0.000],[0.00000002,0.00000004,1.00000000,-0.00000004],[0,-1,0,0],rdkExtax], rdkSpeed, rdkZone, rdkTool, \WObj:=rdkWObj;
	MoveL [[147.288,1945.943,0.000],[0.00000002,0.00000004,1.00000000,-0.00000004],[0,-1,0,0],rdkExtax], rdkSpeed, rdkZone, rdkTool, \WObj:=rdkWObj;
	MoveL [[154.660,1942.009,0.000],[0.00000002,0.00000004,1.00000000,-0.00000004],[0,-1,0,0],rdkExtax], rdkSpeed, rdkZone, rdkTool, \WObj:=rdkWObj;
	MoveL [[161.091,1934.101,0.000],[0.00000002,0.00000004,1.00000000,-0.00000004],[0,-1,0,0],rdkExtax], rdkSpeed, rdkZone, rdkTool, \WObj:=rdkWObj;
	MoveL [[167.817,1923.804,0.000],[0.00000002,0.00000004,1.00000000,-0.00000004],[0,-1,0,0],rdkExtax], rdkSpeed, rdkZone, rdkTool, \WObj:=rdkWObj;
	MoveL [[174.875,1916.208,0.000],[0.00000002,0.00000004,1.00000000,-0.00000004],[0,-1,0,0],rdkExtax], rdkSpeed, rdkZone, rdkTool, \WObj:=rdkWObj;
	MoveL [[182.238,1911.078,0.000],[0.00000002,0.00000004,1.00000000,-0.00000004],[0,-1,0,0],rdkExtax], rdkSpeed, rdkZone, rdkTool, \WObj:=rdkWObj;
	MoveL [[189.879,1908.181,0.000],[0.00000002,0.00000004,1.00000000,-0.00000004],[0,-1,0,0],rdkExtax], rdkSpeed, rdkZone, rdkTool, \WObj:=rdkWObj;
	MoveL [[197.772,1907.282,0.000],[0.00000002,0.00000004,1.00000000,-0.00000004],[0,-1,0,0],rdkExtax], rdkSpeed, rdkZone, rdkTool, \WObj:=rdkWObj;
	MoveL [[205.889,1908.147,0.000],[0.00000002,0.00000004,1.00000000,-0.00000004],[0,-1,0,0],rdkExtax], rdkSpeed, rdkZone, rdkTool, \WObj:=rdkWObj;
	MoveL [[214.204,1910.544,0.000],[0.00000002,0.00000004,1.00000000,-0.00000004],[0,-1,0,0],rdkExtax], rdkSpeed, rdkZone, rdkTool, \WObj:=rdkWObj;
	MoveL [[222.690,1914.236,0.000],[0.00000002,0.00000004,1.00000000,-0.00000004],[0,-1,0,0],rdkExtax], rdkSpeed, rdkZone, rdkTool, \WObj:=rdkWObj;
	MoveL [[231.320,1918.992,0.000],[0.00000002,0.00000004,1.00000000,-0.00000004],[0,-1,0,0],rdkExtax], rdkSpeed, rdkZone, rdkTool, \WObj:=rdkWObj;
	MoveL [[240.067,1924.576,0.000],[0.00000002,0.00000004,1.00000000,-0.00000004],[0,-1,0,0],rdkExtax], rdkSpeed, rdkZone, rdkTool, \WObj:=rdkWObj;
	MoveL [[248.904,1930.754,0.000],[0.00000002,0.00000004,1.00000000,-0.00000004],[0,-1,0,0],rdkExtax], rdkSpeed, rdkZone, rdkTool, \WObj:=rdkWObj;
	MoveL [[257.804,1937.293,0.000],[0.00000002,0.00000004,1.00000000,-0.00000004],[0,-1,0,0],rdkExtax], rdkSpeed, rdkZone, rdkTool, \WObj:=rdkWObj;
	MoveL [[266.741,1943.959,0.000],[0.00000002,0.00000004,1.00000000,-0.00000004],[0,-1,0,0],rdkExtax], rdkSpeed, rdkZone, rdkTool, \WObj:=rdkWObj;
	MoveL [[275.687,1950.518,0.000],[0.00000002,0.00000004,1.00000000,-0.00000004],[0,-1,0,0],rdkExtax], rdkSpeed, rdkZone, rdkTool, \WObj:=rdkWObj;
	MoveL [[284.616,1956.735,0.000],[0.00000002,0.00000004,1.00000000,-0.00000004],[0,-1,0,0],rdkExtax], rdkSpeed, rdkZone, rdkTool, \WObj:=rdkWObj;
	MoveL [[293.501,1962.377,0.000],[0.00000002,0.00000004,1.00000000,-0.00000004],[0,-1,0,0],rdkExtax], rdkSpeed, rdkZone, rdkTool, \WObj:=rdkWObj;
	MoveL [[302.315,1967.210,0.000],[0.00000002,0.00000004,1.00000000,-0.00000004],[0,-1,0,0],rdkExtax], rdkSpeed, rdkZone, rdkTool, \WObj:=rdkWObj;
	MoveL [[311.031,1970.999,0.000],[0.00000002,0.00000004,1.00000000,-0.00000004],[0,-1,0,0],rdkExtax], rdkSpeed, rdkZone, rdkTool, \WObj:=rdkWObj;
	MoveL [[319.752,1975.169,0.000],[0.00000002,0.00000004,1.00000000,-0.00000004],[0,-1,0,0],rdkExtax], rdkSpeed, rdkZone, rdkTool, \WObj:=rdkWObj;
	MoveL [[328.504,1980.131,0.000],[0.00000002,0.00000004,1.00000000,-0.00000004],[0,-1,0,0],rdkExtax], rdkSpeed, rdkZone, rdkTool, \WObj:=rdkWObj;
	MoveL [[337.301,1985.071,0.000],[0.00000002,0.00000004,1.00000000,-0.00000004],[0,-1,0,0],rdkExtax], rdkSpeed, rdkZone, rdkTool, \WObj:=rdkWObj;
	MoveL [[346.217,1989.767,0.000],[0.00000002,0.00000004,1.00000000,-0.00000004],[0,-1,0,0],rdkExtax], rdkSpeed, rdkZone, rdkTool, \WObj:=rdkWObj;
	MoveL [[355.322,1993.994,0.000],[0.00000002,0.00000004,1.00000000,-0.00000004],[0,-1,0,0],rdkExtax], rdkSpeed, rdkZone, rdkTool, \WObj:=rdkWObj;
	MoveL [[364.689,1997.529,0.000],[0.00000002,0.00000004,1.00000000,-0.00000004],[0,-1,0,0],rdkExtax], rdkSpeed, rdkZone, rdkTool, \WObj:=rdkWObj;
	MoveL [[374.392,2000.149,0.000],[0.00000002,0.00000004,1.00000000,-0.00000004],[0,-1,0,0],rdkExtax], rdkSpeed, rdkZone, rdkTool, \WObj:=rdkWObj;
	MoveL [[374.392,2000.149,100.000],[0.00000002,0.00000004,1.00000000,-0.00000004],[0,-1,0,0],rdkExtax], rdkSpeed, rdkZone, rdkTool, \WObj:=rdkWObj;
	MoveL CalcRobT([[0.000000,0.000000,0.000000,0.000000,90.000000,0.000000],rdkExtax], rdkTool \WObj:=rdkWObj), rdkSpeed, rdkZone, rdkTool, \WObj:=rdkWObj;
ENDPROC

ENDMODULE
